Yaskawa INFORM job: ARUBA_2.JBI

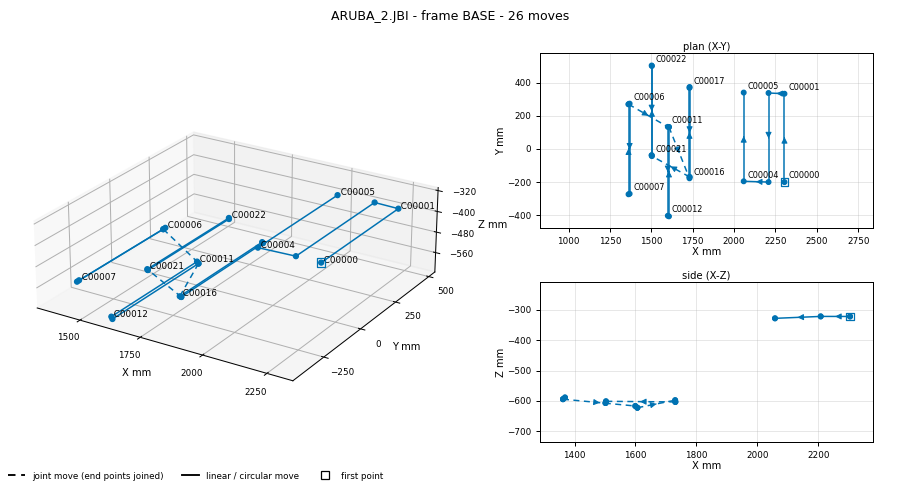
[picture p0: tool path of ARUBA_2.JBI in frame BASE, 26 of 32 moves have a stored position in this frame; points joined in program order, loops and branches not executed]
/JOB
//NAME ARUBA_2
//POS
///NPOS 26,0,26,0,0,0
///TOOL 0
///POSTYPE BASE
///RECTAN
///RCONF 1,0,0,0,0,0,0,0,0,0,0,0,0,0,0,0,0,0,0,0,0,0,0,0
C00000=2304.322058,-200.343917,-322.557006,175.000000,5.000000,5.000000
C00001=2304.322058,333.611356,-322.557006,175.000000,5.000000,5.000000
C00002=2208.055638,338.026842,-322.379244,175.000000,5.000000,5.000000
C00003=2208.055638,-200.236990,-322.379244,175.000000,5.000000,5.000000
C00004=2058.014577,-195.577258,-328.715056,175.000000,5.000000,5.000000
C00005=2058.014577,340.670714,-328.715056,175.000000,5.000000,5.000000
C00006=1368.622502,273.835769,-588.454909,175.000000,-89.999999,5.000000
C00007=1368.622502,-270.904268,-588.454909,175.000000,-89.999999,5.000000
C00008=1362.058578,-274.148687,-594.117341,180.000000,-60.000000,0.000000
C00009=1362.058578,269.992267,-594.117341,180.000000,-60.000000,0.000000
C00010=1362.058578,269.992267,-594.117341,180.000000,-60.000000,0.000000
C00011=1599.399476,133.522218,-616.439062,175.000000,-89.999999,5.000000
C00012=1599.399476,-403.921612,-616.439062,175.000000,-89.999999,5.000000
C00013=1606.255755,-407.412419,-622.101494,180.000000,-60.000000,0.000000
C00014=1606.255755,132.326729,-622.101494,180.000000,-60.000000,0.000000
C00015=1606.255755,132.326729,-622.101494,180.000000,-60.000000,0.000000
C00016=1730.321934,-177.566018,-597.423267,175.000000,-89.999999,5.000000
C00017=1730.321934,369.090460,-597.423267,175.000000,-89.999999,5.000000
C00018=1730.927977,374.284826,-603.085699,180.000000,-60.000000,0.000000
C00019=1730.927977,-169.242399,-603.085699,180.000000,-60.000000,0.000000
C00020=1730.927977,-169.242399,-603.085699,180.000000,-60.000000,0.000000
C00021=1503.225343,-43.528433,-601.036284,175.000000,-89.999999,5.000000
C00022=1503.225343,501.238678,-601.036284,175.000000,-89.999999,5.000000
C00023=1501.802779,504.032955,-606.698717,180.000000,-60.000000,0.000000
C00024=1501.802779,-38.254983,-606.698717,180.000000,-60.000000,0.000000
C00025=1501.802779,-38.254983,-606.698717,180.000000,-60.000000,0.000000
///POSTYPE PULSE
///PULSE
EC00000=0
EC00001=0
EC00002=0
EC00003=0
EC00004=0
EC00005=0
EC00006=0
EC00007=0
EC00008=0
EC00009=0
EC00010=92160
EC00011=92160
EC00012=92160
EC00013=92160
EC00014=92160
EC00015=184320
EC00016=184320
EC00017=184320
EC00018=184320
EC00019=184320
EC00020=276480
EC00021=276480
EC00022=276480
EC00023=276480
EC00024=276480
EC00025=368640
//INST
///DATE 2023/05/05 17:53
///ATTR SC,RW,RJ
////FRAME BASE
///GROUP1 RB1,ST1
NOP
MOVJ P009 EX000 VJ=15.00
MOVJ C00000 EC00000 VJ=15.0
CALL JOB:SPYON
MOVL C00001 EC00001 V=200.0
MOVL C00002 EC00002 V=200.0
MOVL C00003 EC00003 V=200.0
MOVL C00004 EC00004 V=200.0
MOVL C00005 EC00005 V=200.0
CALL JOB:SPYOF
MOVJ P009 VJ=15.00
MOVJ C00006 EC00006 VJ=15.0
CALL JOB:SPYON
MOVL C00007 EC00007 V=200.0
MOVL C00008 EC00008 V=200.0
MOVL C00009 EC00009 V=200.0
CALL JOB:SPYOF
MOVJ P009 VJ=15.00
MOVL C00010 EC00010 V=200.0
MOVJ C00011 EC00011 VJ=15.0
CALL JOB:SPYON
MOVL C00012 EC00012 V=200.0
MOVL C00013 EC00013 V=200.0
MOVL C00014 EC00014 V=200.0
CALL JOB:SPYOF
MOVJ P009 VJ=15.00
MOVL C00015 EC00015 V=200.0
MOVJ C00016 EC00016 VJ=15.0
CALL JOB:SPYON
MOVL C00017 EC00017 V=200.0
MOVL C00018 EC00018 V=200.0
MOVL C00019 EC00019 V=200.0
CALL JOB:SPYOF
MOVJ P009 VJ=15.00
MOVL C00020 EC00020 V=200.0
MOVJ C00021 EC00021 VJ=15.0
CALL JOB:SPYON
MOVL C00022 EC00022 V=200.0
MOVL C00023 EC00023 V=200.0
MOVL C00024 EC00024 V=200.0
CALL JOB:SPYOF
MOVJ P009 VJ=15.00
MOVL C00025 EC00025 V=200.0
END
